SUBAPPLICATION Knickdeichsel (* Subapplication Type *)
  (* Standard: 61499-2 *)
  (* Version 1.0, 2023-01-29, Franz *)
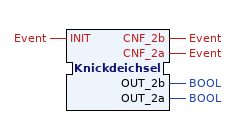
  EVENT_INPUT
    INIT;
  END_EVENT
  EVENT_OUTPUT
    CNF_2b;
    CNF_2a;
  END_EVENT
  VAR_OUTPUT
    OUT_2b : BOOL;
    OUT_2a : BOOL;
  END_VAR
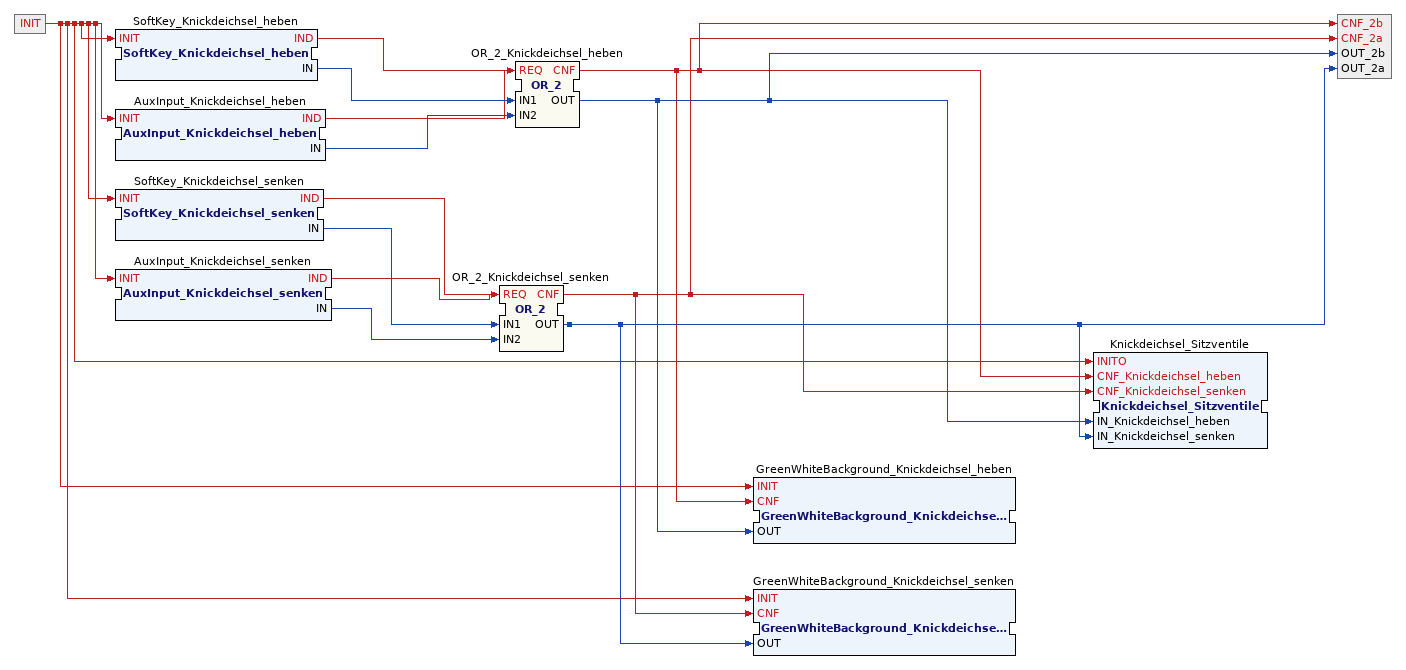
  FBS
    OR_2_Knickdeichsel_heben : OR_2;
    OR_2_Knickdeichsel_senken : OR_2;
  END_FBS
  SUBAPPS
    GreenWhiteBackground_Knickdeichsel_heben : GreenWhiteBackground_Knickdeichsel_heben;
    GreenWhiteBackground_Knickdeichsel_senken : GreenWhiteBackground_Knickdeichsel_senken;
    Knickdeichsel_Sitzventile : Knickdeichsel_Sitzventile;
    SoftKey_Knickdeichsel_heben : SoftKey_Knickdeichsel_heben;
    SoftKey_Knickdeichsel_senken : SoftKey_Knickdeichsel_senken;
    AuxInput_Knickdeichsel_senken : AuxInput_Knickdeichsel_senken;
    AuxInput_Knickdeichsel_heben : AuxInput_Knickdeichsel_heben;
  END_SUBAPPS
  EVENT_CONNECTIONS
    INIT TO GreenWhiteBackground_Knickdeichsel_heben.INIT;
    INIT TO GreenWhiteBackground_Knickdeichsel_senken.INIT;
    INIT TO Knickdeichsel_Sitzventile.INITO;
    INIT TO SoftKey_Knickdeichsel_heben.INIT;
    INIT TO SoftKey_Knickdeichsel_senken.INIT;
    INIT TO AuxInput_Knickdeichsel_senken.INIT;
    SoftKey_Knickdeichsel_heben.IND TO OR_2_Knickdeichsel_heben.REQ;
    OR_2_Knickdeichsel_heben.CNF TO GreenWhiteBackground_Knickdeichsel_heben.CNF;
    OR_2_Knickdeichsel_heben.CNF TO Knickdeichsel_Sitzventile.CNF_Knickdeichsel_heben;
    SoftKey_Knickdeichsel_senken.IND TO OR_2_Knickdeichsel_senken.REQ;
    AuxInput_Knickdeichsel_senken.IND TO OR_2_Knickdeichsel_senken.REQ;
    OR_2_Knickdeichsel_senken.CNF TO GreenWhiteBackground_Knickdeichsel_senken.CNF;
    OR_2_Knickdeichsel_senken.CNF TO Knickdeichsel_Sitzventile.CNF_Knickdeichsel_senken;
    INIT TO AuxInput_Knickdeichsel_heben.INIT;
    AuxInput_Knickdeichsel_heben.IND TO OR_2_Knickdeichsel_heben.REQ;
    OR_2_Knickdeichsel_heben.CNF TO CNF_2b;
    OR_2_Knickdeichsel_senken.CNF TO CNF_2a;
  END_CONNECTIONS
  DATA_CONNECTIONS
    SoftKey_Knickdeichsel_heben.IN TO OR_2_Knickdeichsel_heben.IN1;
    OR_2_Knickdeichsel_heben.OUT TO GreenWhiteBackground_Knickdeichsel_heben.OUT;
    OR_2_Knickdeichsel_heben.OUT TO Knickdeichsel_Sitzventile.IN_Knickdeichsel_heben;
    SoftKey_Knickdeichsel_senken.IN TO OR_2_Knickdeichsel_senken.IN1;
    AuxInput_Knickdeichsel_senken.IN TO OR_2_Knickdeichsel_senken.IN2;
    OR_2_Knickdeichsel_senken.OUT TO GreenWhiteBackground_Knickdeichsel_senken.OUT;
    OR_2_Knickdeichsel_senken.OUT TO Knickdeichsel_Sitzventile.IN_Knickdeichsel_senken;
    AuxInput_Knickdeichsel_heben.IN TO OR_2_Knickdeichsel_heben.IN2;
    OR_2_Knickdeichsel_heben.OUT TO OUT_2b;
    OR_2_Knickdeichsel_senken.OUT TO OUT_2a;
  END_CONNECTIONS
END_SUBAPPLICATION
